RoboDK station: UR3_Simulate.rdk

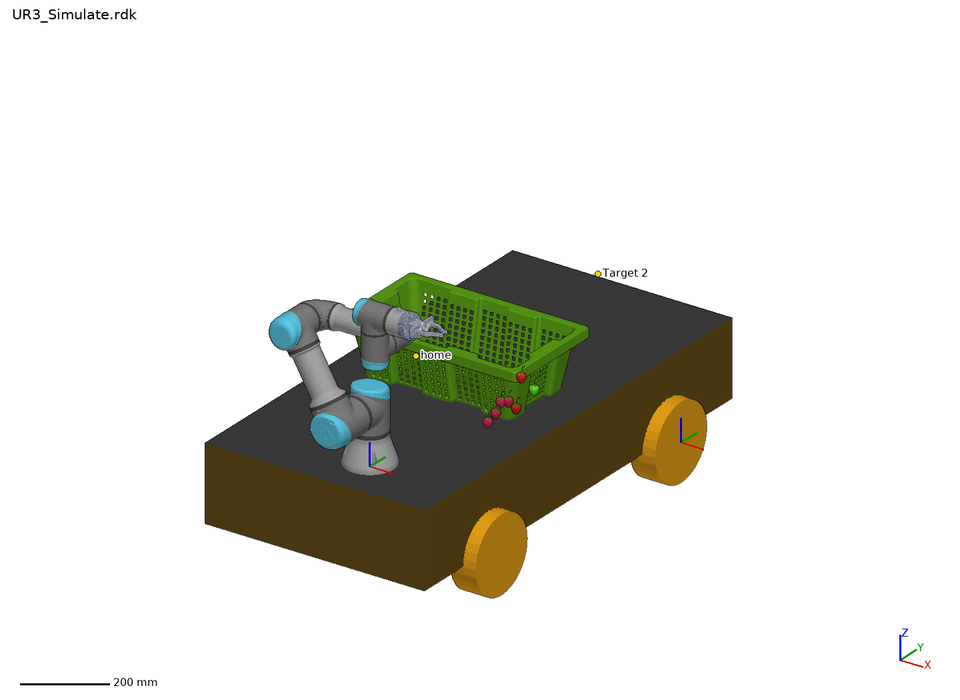
[picture v0: the station drawn from its stored meshes, robots at their saved joint values, targets as dots, program paths as lines]
Station UR3_Simulate (saved by RoboDK 5.6.3). Poses are relative to the parent item; angles as X-Y-Z fixed-axis rotations.
  - frame UR3 Base at (0, 0, 0) mm
    - robot UR3: 6 axes, payload 3 kg, reach 500 mm, repeatability 0.1 mm, weight 11 kg
        modified DH rows (alpha deg, a mm, theta deg, d mm): 0, 0, 0, 151.9; 90, 0, 180, 0; 0, 243.65, 0, 0; 0, 213, 0, 110.4; -90, 0, 0, 83.4; 90, 0, 180, 82.4
        joint limits [-360, -360, -360, -360, -360, -360] to [360, 360, 360, 360, 360, 360]; home [0, -90, -90, 0, 90, 0]; saved at [0, -60, -120, 0, 90, 0]
      - tool Tool 1, TCP at (0, 70, 30) mm
      - tool Tool_Assem, TCP at (-3.5, 6, 93) mm, size 88 x 65 x 108.8 mm, geometry from Tool_Assem.IGS
    - frame Reference SW at (500, 500, 0) mm
      - object Strawberry_Red_1 at (-10, -610, 400) mm, rotated rx 90 ry 0 rz 0 deg, size 22.9 x 39 x 26.9 mm, geometry from SB-Strawberry.IGS
      - object Base at (-560, -30, -190) mm, rotated rx 90 ry 0 rz 90 deg, size 1200 x 300 x 670 mm, geometry from Base.IGS
      - object Strawberry_Green at (-10, -560, 350) mm, rotated rx 90 ry 0 rz 0 deg, size 22.9 x 39 x 26.9 mm, geometry from SB-Strawberry.IGS
      - object plastic bucket 2 at (-560, -50, 12) mm, rotated rx 90 ry 0 rz 0 deg, size 490 x 153 x 290 mm, geometry from plastic bucket 2.IGS
      - object Strawberry_Red_2 at (-10, -660, 360) mm, rotated rx 90 ry 0 rz 0 deg, size 22.9 x 39 x 26.9 mm, geometry from SB-Strawberry.IGS
      - object Strawberry_Red_3 at (-10, -630, 330) mm, rotated rx 90 ry 0 rz 0 deg, size 22.9 x 39 x 26.9 mm, geometry from SB-Strawberry.IGS
      - object Strawberry_Red_4 at (-10, -690, 370) mm, rotated rx 90 ry 0 rz 0 deg, size 22.9 x 39 x 26.9 mm, geometry from SB-Strawberry.IGS
      - object Strawberry_Red_5 at (-10, -710, 350) mm, rotated rx 90 ry 0 rz 0 deg, size 22.9 x 39 x 26.9 mm, geometry from SB-Strawberry.IGS
      - object Strawberry_Red_6 at (-10, -740, 340) mm, rotated rx 90 ry 0 rz 0 deg, size 22.9 x 39 x 26.9 mm, geometry from SB-Strawberry.IGS
    - target home (joint target) at (203.57, -110.4, 376.31) mm, rotated rx -90 ry 0 rz -90 deg; joints [0, -60, -120, 0, 90, 0] of UR3
    - target Target 2 (Cartesian target) at (491.75, 186, 543) mm, rotated rx -90 ry 0 rz -90 deg; joints [28.399, -139.214, -12.222, -28.564, 61.601, 0] of UR3
  - camera Camera 1
  - program Prog1 (1 instructions, listed below)

--- program Prog1 (robot UR3) ---
  Set speed (30.0 mm/s)
